PROGRAM MAIN
VAR
END_VAR

M_SING();
M_MOTOR();

METHOD M_MOTOR : BOOL
VAR_INPUT
END_VAR
gvl.bmotorcontrol := ((gvl.bmotorstartpb or gvl.bmotorcontrol) and (not gvl.bmotorstoppb) ) and gvl.bmotorcontrolenable;

//	GVL.bmotorstartpb := false;
//	gvl.bmotorstoppb := false;
END_METHOD

METHOD M_SING : BOOL
VAR_INPUT
END_VAR


GVL.RX 		:= 0.02 + GVL.rX;

IF GVL.rY > (3.14 * 2.0) THEN
	
	GVL.RX := 0;
	
END_IF
GVL.rY  	:= SIN(GVL.RX);
END_METHOD

END_PROGRAM

(* stored: Version 1.1.0.1, ProductVersion 3.1.4024.12
   POU MAIN: Id {370f09e1-aab9-4631-a45b-98d4087e384f}, SpecialFunc None
   Method M_MOTOR: Id {59edf82d-8b44-427b-bf27-2b34876429cb}
   Method M_SING: Id {980af3c3-0c25-4c01-b933-580ca6d36e12} *)
